FUNCTION_BLOCK RemoveAMover_TestSuite
VAR
	ThisTestSuite : TestSuite<TestSuiteParameter.MaxTestCount>('C:\ProgramData\Beckhoff\TwinCAT\3.1\Boot\RemoveSingle_Tests.xml') := (TestSuiteName := 'RemoveSingle Test Suite');
END_VAR

TaskAcceptsRemoveCommand();
TaskRejectsDuplicatecommand_Test();
TaskRejectsCycleWithNoGroup_Test();
TaskRejectsExecuteWithNoGroup_Test();
TaskRejectsInvalidCAGroup();

METHOD TaskAcceptsRemoveCommand
VAR
	stubGroup : CollisionGroup;
	testRemoveAMover : RemoveMoverFromGroup :=(MyCollisionGroup := stubGroup);
	Expected : BOOL := TRUE;
	Actual	 : BOOL;
END_VAR
IF ThisTestSuite.Test(__POUNAME()).ExecuteTest() THEN
	Actual := SUCCEEDED(testRemoveAMover.Execute(AxisID := UDINT_TO_IDENTINGROUP(2)));
	ThisTestSuite.Test(__POUNAME()).AssertEqual(Expected, Actual);
END_IF
END_METHOD

METHOD TaskRejectsCycleWithNoGroup_Test
VAR
	testRemoveAMover : RemoveMoverFromGroup;
	Expected : BOOL := TRUE;
	Actual	 : BOOL;
END_VAR
IF ThisTestSuite.Test(__POUNAME()).ExecuteTest() THEN
	Actual := failed(testRemoveAMover.Cycle());
	ThisTestSuite.Test(__POUNAME()).AssertEqual(Expected, Actual);
END_IF
END_METHOD

METHOD TaskRejectsDuplicatecommand_Test
VAR
	stubGroup : CollisionGroup;
	testRemoveAMover : RemoveMoverFromGroup :=(MyCollisionGroup := stubGroup);
	Expected : BOOL := TRUE;
	Actual	 : BOOL;
END_VAR
IF ThisTestSuite.Test(__POUNAME()).ExecuteTest() THEN
	testRemoveAMover.Execute(AxisID := UDINT_TO_IDENTINGROUP(2));
	Actual := FAILED(testRemoveAMover.Execute(AxisID := UDINT_TO_IDENTINGROUP(2)));
	ThisTestSuite.Test(__POUNAME()).AssertEqual(Expected, Actual);
END_IF
END_METHOD

METHOD TaskRejectsExecuteWithNoGroup_Test
VAR
	testRemoveAMover : RemoveMoverFromGroup;
	Expected : BOOL := TRUE;
	Actual	 : BOOL;
END_VAR
IF ThisTestSuite.Test(__POUNAME()).ExecuteTest() THEN
	Actual := failed(testRemoveAMover.Execute(AxisID := UDINT_TO_IDENTINGROUP(2)));
	ThisTestSuite.Test(__POUNAME()).AssertEqual(Expected, Actual);
END_IF
END_METHOD

METHOD TaskRejectsInvalidCAGroup
VAR
	stubGroup : CollisionGroup;
	iStubCAGRoup : I_CollisionGroup := stubGroup;
	testRemoveAMover : RemoveMoverFromGroup :=(MyCollisionGroup := stubGroup);
	Expected : BOOL := TRUE;
	Actual	 : BOOL;
END_VAR
IF ThisTestSuite.Test(__POUNAME()).ExecuteTest() THEN
	testRemoveAMover.MyCollisionGroup := 16#0;
	Actual := testRemoveAMover.MyCollisionGroup = iStubCAGroup;
	ThisTestSuite.Test(__POUNAME()).AssertEqual(Expected, Actual);
END_IF
END_METHOD

END_FUNCTION_BLOCK

(* stored: Version 1.1.0.1
   POU RemoveAMover_TestSuite: Id {073eca12-f7a7-4609-978a-c4fbddc5e48d}, SpecialFunc None
   Method TaskAcceptsRemoveCommand: Id {9701816a-7347-4094-8354-4a80b2556129}
   Method TaskRejectsCycleWithNoGroup_Test: Id {65ff5eec-b310-4399-b6c7-df2c2d9aab4b}
   Method TaskRejectsDuplicatecommand_Test: Id {b24cbb70-1da5-46eb-b97d-f92f9948b290}
   Method TaskRejectsExecuteWithNoGroup_Test: Id {2bc3b776-9613-4a5b-bf0e-583ff32a2592}
   Method TaskRejectsInvalidCAGroup: Id {a95a7c96-c991-4b11-9d40-aa3626e3c936} *)
